TYPE (* IEC61131-3, Table 14#5 *)
  (* Standard: 1131-3 *)
  (* Version 0.0, 1/8/2024, Cheyan, Schneider Electric, Template *)
  PACKAGE Main;
  {SET_ATTRIBUTE(nxtDataType, 9gA4evvp0K20hxdCgULQYkV6QmDNh3dwMc8Ym4KvG+kuAJ0VWwsPMcE01ZsquGuVqZAGwyjk+Pz/7Ur1FoSLmjuJQJnqKPem17tDavdvsGG6DhN/811gPwZegzo+YN9HE8GC5JrPj89E8RyObJA/iMWQ12cACnhJ1pctbom+kjmWIgMIr5gHpdsh7tVoZWMTRvBOhWhLyLIQDIo8tB1BUys1QUlkfiGc)}
  SPS_BOOL : STRUCT
    stVal : BOOL;
    q : Quality;
    t : TimeStamp;
  END_STRUCT;
END_TYPE
